(* PLC project Unnamed, Unknown Unnamed 1 *)
(* stored: creationDateTime 2025-04-06T18:12:44, modificationDateTime 2025-04-06T22:26:21 *)

PROGRAM program0
  VAR
    St0 : BOOL := 1;
    St1 : BOOL := 0;
    St2 : BOOL := 0;
  END_VAR
  VAR
    B1 AT %IX0.0 : BOOL := 0;
    B2 AT %IX0.1 : BOOL := 0;
    B3 AT %IX0.2 : BOOL := 0;
    DC AT %QX0.2 : BOOL := 0;
  END_VAR
  VAR
    StepDone : BOOL;
  END_VAR
  VAR
    StepRun AT %QX0.1 : BOOL;
  END_VAR
  VAR
    TON0 : TON;
  END_VAR

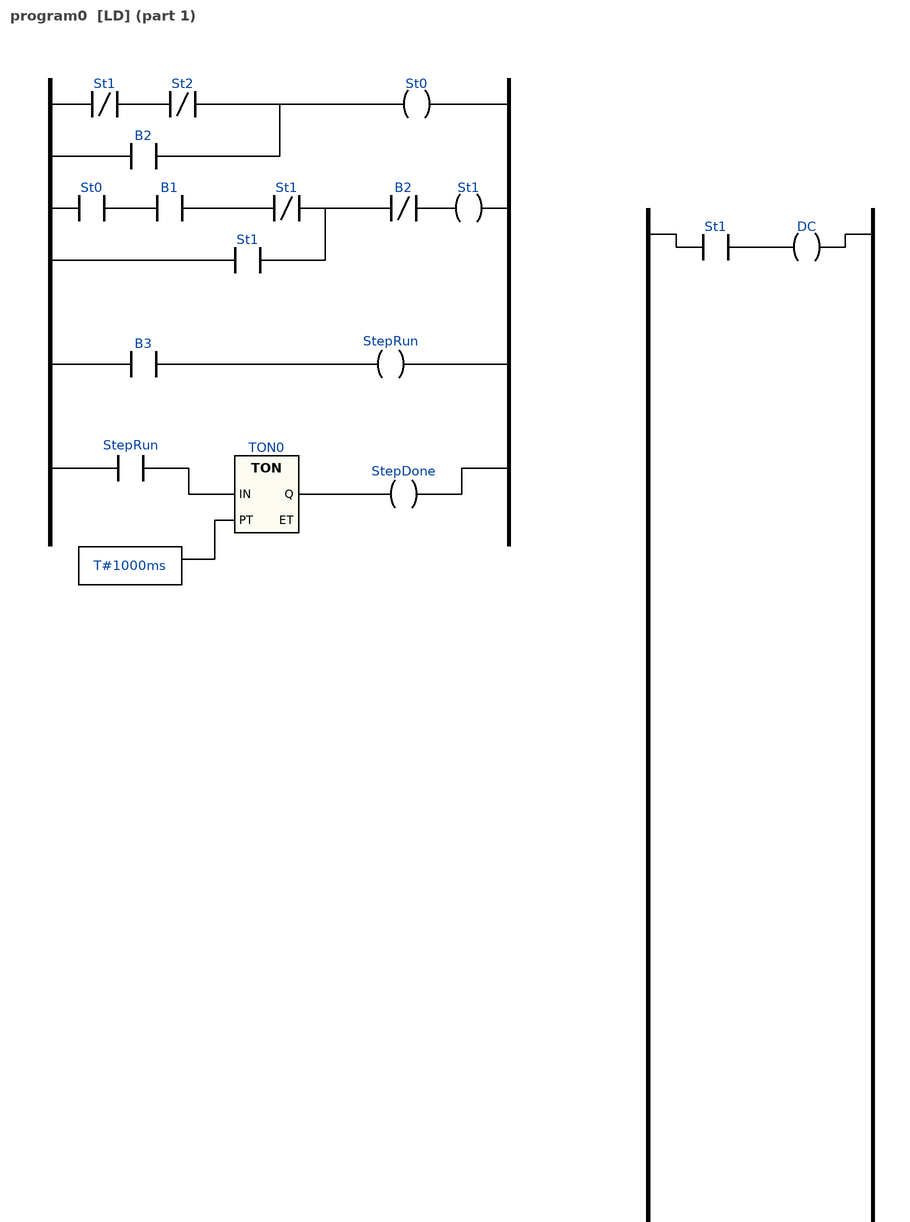
(* LD diagram, written out as Structured Text *)
St0 := NOT St1 AND NOT St2 OR B2;
St1 := (St1 OR St0 AND B1 AND NOT St1) AND NOT B2;
StepRun := B3;
TON0(IN := StepRun, PT := T#1000ms);
StepDone := TON0.Q;
DC := St1;
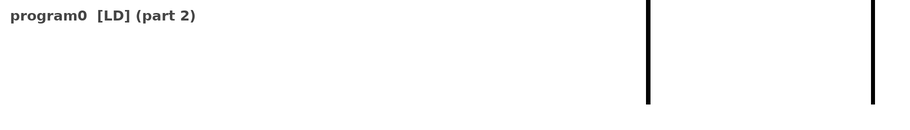
END_PROGRAM

CONFIGURATION Config0
  RESOURCE Res0 ON PLC
    TASK task0(INTERVAL := T#20ms, PRIORITY := 0);
    PROGRAM instance0 WITH task0 : program0;
  END_RESOURCE
END_CONFIGURATION
